// TIA Portal project "5 Run - 2 Stop For 2 Motors" (V16)

(* hardware
DEVICE "S7-1200 station_1"  S7-1200 Station
   slot 0: "Rack_0"  S7-1200 Rack  Rack  V1.0
   slot 1: "PLC_1"  CPU 1212C AC/DC/Rly  6ES7 212-1BE40-0XB0  V4.0
*)

// ===== PLC "PLC_1"  CPU 1212C AC/DC/Rly =====

VAR_GLOBAL   // PLC tag table "Default tag table"
   "start1" AT %I0.2 : Bool;
   "K1" AT %Q0.0 : Bool;
   "stop1" AT %I0.4 : Bool;
   "k2" AT %Q0.1 : Bool;
   "start2" AT %I0.3 : Bool;
   "T1 tag" AT %M0.0 : Bool;
   "T2 tag" AT %M0.1 : Bool;
   "X" AT %M0.2 : Bool;
   "C1 TAG" AT %M0.3 : Bool;
   "T2 COUNT tag" AT %M0.4 : Bool;
   "T3 tag" AT %M0.7 : Bool;
   "k2 tag" AT %M1.4 : Bool;
   "k1<>k2" AT %M5.0 : Bool;
   "T3 tag(1)" AT %M3.0 : Bool;
   "T4 tag" AT %M1.0 : Bool;
   "Tag_3" AT %M3.5 : Bool;
   "C2 tag" AT %M1.2 : Bool;
   "T4 COUNT tag" AT %M1.5 : Bool;
   "K1 stopped 2S" AT %M8.0 : Bool;
END_VAR

// folder: System blocks/Program resources

DATA_BLOCK "T2"   // DB1
{ S7_Optimized_Access := 'TRUE' }
AUTHOR : Simatic
FAMILY : IEC
NAME : IEC_TMR
VERSION : 1.0
// stored: InstanceOfName IEC_TIMER
"IEC_TIMER"
BEGIN
END_DATA_BLOCK

DATA_BLOCK "T1"   // DB2
{ S7_Optimized_Access := 'TRUE' }
AUTHOR : Simatic
FAMILY : IEC
NAME : IEC_TMR
VERSION : 1.0
// stored: InstanceOfName IEC_TIMER
"IEC_TIMER"
BEGIN
END_DATA_BLOCK

DATA_BLOCK "C1"   // DB3
{ S7_Optimized_Access := 'TRUE' }
AUTHOR : Simatic
FAMILY : IEC
NAME : CNTR
VERSION : 1.0
// stored: InstanceOfName IEC_COUNTER
"IEC_COUNTER"
BEGIN
END_DATA_BLOCK

DATA_BLOCK "T3"   // DB4
{ S7_Optimized_Access := 'TRUE' }
AUTHOR : Simatic
FAMILY : IEC
NAME : IEC_TMR
VERSION : 1.0
// stored: InstanceOfName IEC_TIMER
"IEC_TIMER"
BEGIN
END_DATA_BLOCK

DATA_BLOCK "T4"   // DB5
{ S7_Optimized_Access := 'TRUE' }
AUTHOR : Simatic
FAMILY : IEC
NAME : IEC_TMR
VERSION : 1.0
// stored: InstanceOfName IEC_TIMER
"IEC_TIMER"
BEGIN
END_DATA_BLOCK

DATA_BLOCK "C2"   // DB6
{ S7_Optimized_Access := 'TRUE' }
AUTHOR : Simatic
FAMILY : IEC
NAME : CNTR
VERSION : 1.0
// stored: InstanceOfName IEC_COUNTER
"IEC_COUNTER"
BEGIN
END_DATA_BLOCK

// folder: (top level)

ORGANIZATION_BLOCK "Main"   // OB1, LAD, ProgramCycle
TITLE = "Main Program Sweep (Cycle)"
{ S7_Optimized_Access := 'TRUE' }
VERSION : 0.1
   VAR_INPUT
      Initial_Call : Bool;   // Initial call of this OB
      Remanence : Bool;   // =True, if remanent data are available
   END_VAR
   VAR_TEMP   // added for the SCL form of the ladder/FBD networks
      _w1 : Bool;
   END_VAR
BEGIN

REGION Network 1: start
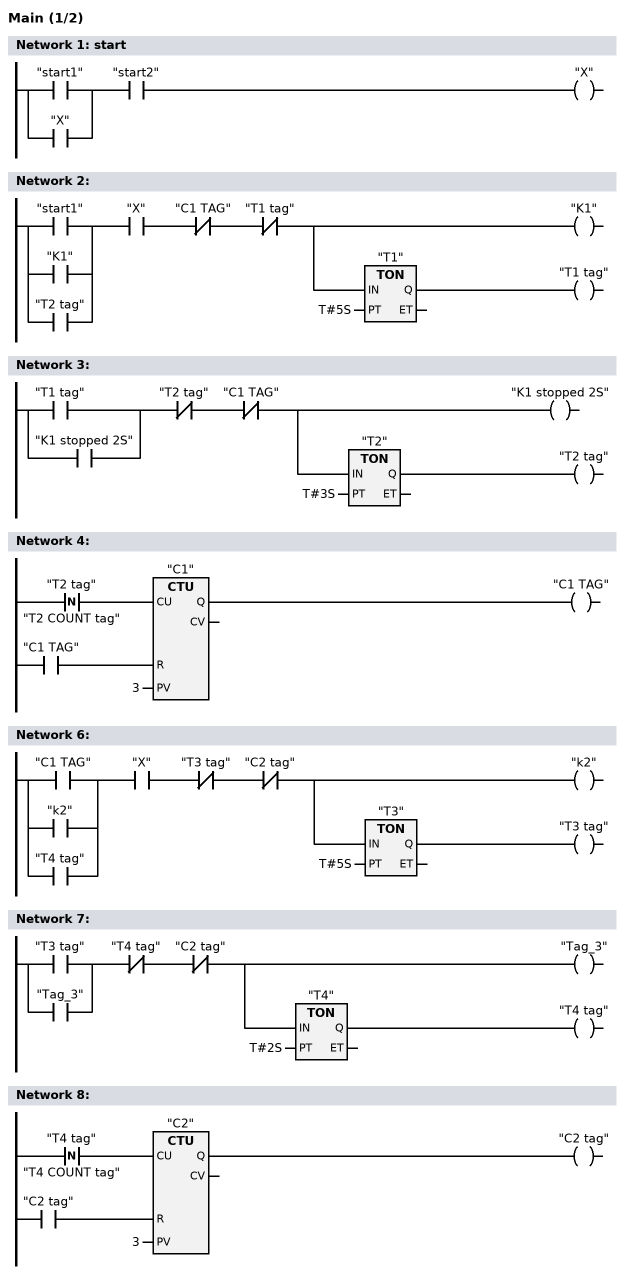
   RUNG wire#powerrail
      Contact( "start1" )
      wire#w1
      Contact( "start2" )
      Coil( "X" )
   END_RUNG
   RUNG wire#powerrail
      Contact( "X" )
   END_RUNG wire#w1
   // the same network as SCL:
   "X" := ("start1" OR "X") AND "start2";
END_REGION

REGION Network 2
   "K1" := ("start1" OR "K1" OR "T2 tag") AND "X" AND NOT "C1 TAG" AND NOT "T1 tag";
   "T1".TON(IN := "K1", PT := T#5S);
   "T1 tag" := "T1".Q;
END_REGION

REGION Network 3
   "K1 stopped 2S" := ("T1 tag" OR "K1 stopped 2S") AND NOT "T2 tag" AND NOT "C1 TAG";
   "T2".TON(IN := "K1 stopped 2S", PT := T#3S);
   "T2 tag" := "T2".Q;
END_REGION

REGION Network 4
   #_w1 := NOT "T2 tag" AND "T2 COUNT tag";   // falling edge of "T2 tag"
   "T2 COUNT tag" := "T2 tag";
   "C1".CTU(CU := #_w1, R := "C1 TAG", PV := 3);
   "C1 TAG" := "C1".Q;
END_REGION

REGION Network 6
   "k2" := ("C1 TAG" OR "k2" OR "T4 tag") AND "X" AND NOT "T3 tag" AND NOT "C2 tag";
   "T3".TON(IN := "k2", PT := T#5S);
   "T3 tag" := "T3".Q;
END_REGION

REGION Network 7
   "Tag_3" := ("T3 tag" OR "Tag_3") AND NOT "T4 tag" AND NOT "C2 tag";
   "T4".TON(IN := "Tag_3", PT := T#2S);
   "T4 tag" := "T4".Q;
END_REGION

REGION Network 8
   #_w1 := NOT "T4 tag" AND "T4 COUNT tag";   // falling edge of "T4 tag"
   "T4 COUNT tag" := "T4 tag";
   "C2".CTU(CU := #_w1, R := "C2 tag", PV := 3);
   "C2 tag" := "C2".Q;
END_REGION

REGION Network 9
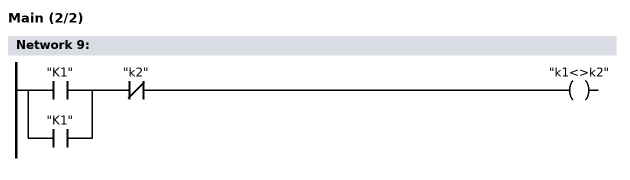
   RUNG wire#powerrail
      Contact( "K1" )
      wire#w1
      I_Contact( "k2" )
      Coil( "k1<>k2" )
   END_RUNG
   RUNG wire#powerrail
      Contact( "K1" )
   END_RUNG wire#w1
   // the same network as SCL:
   "k1<>k2" := ("K1" OR "K1") AND NOT "k2";
END_REGION
END_ORGANIZATION_BLOCK